Fanuc KAREL source: COPY_PATH.kl

PROGRAM T
%NOLOCKGROUP
VAR
 v0 : PATH
 v1 : INTEGER
 v2 : INTEGER
 v3 : PATH
 v4 : INTEGER
BEGIN
 COPY_PATH(v0, v1, v2, v3, v4)
END T
